Staubli VAL3: stopExtAxis.pgx

public program stopExtAxis(num x_nAxisNum)
begin
  //
  if blifebit[x_nAxisNum]
    doQuickStop[x_nAxisNum]=false
    doSwitchOn[x_nAxisNum]=false
    doEnableVoltage[x_nAxisNum]=false
    doEnableOp[x_nAxisNum]=false
    doStartHoming[x_nAxisNum]=false
    aioSet(aoWorkMode[x_nAxisNum],0)
  endIf
end
